{attribute 'no_check'}
// ModBus comunication master to multible slaves useing RTU protocol
// based on TF6255 - required lib: Tc2_ModbusRTU
FUNCTION_BLOCK ModbusRtuMaster22B
VAR_OUTPUT CONSTANT
	MIN_SLAVE												:	INT := 1;
	MAX_SLAVE												:	INT := PARAM.MODBUS_MAX_SLAVES_OF_MASTER;
{attribute 'displaymode':='binary'}
	OPTION_DISABLE_ERROR_STATE								:	BYTE := 2#0000_0001; //FB will not go into error state and keeps running, even all slaves are in error state
END_VAR
VAR_INPUT
	Enable													:	BOOL ; 		// FB will be processed as long as enable is TRUE 
	ResetTrig												:	BOOL ;		// The function block will be reset with a rising edge 
{attribute 'displaymode':='binary'}
	Options													:	BYTE := 0; //FB options, see VAR_OUTPUT CONSTANT
	SlaveCom												:	ARRAY[MIN_SLAVE..MAX_SLAVE] OF POINTER TO ModbusSlaveCom;
	Timestamp												:	DT;
END_VAR         	
VAR_OUTPUT     
	JobNo													:	INT := 0;
	SlaveNo													:	INT := 0;
{attribute 'displaymode':='binary'}
	SlaveInErrorMask										:	DWORD; //Bit.1 indicates slave 1 in error 	
	Error													:	BOOL;		// Rising edge of Error informs that an error occurred during the execution of the Function Block 
{attribute 'displaymode':='hex'}
	ErrorID													:	MODBUS_ERRORS;		// Error identification - see ADS return codes at Beckhoff infosys for further information 
	ErrorText												:	STRING;
END_VAR
VAR
(* memory **************************************************)
	State 													:	INT := 0;
(* trigger *************************************************)

(* timer ***************************************************)

(* blocks **************************************************)
//	com														:	ModbusRtuMaster_PcCOM := (Timeout := DEFAULT_ADS_TIMEOUT);
	com														:	ModbusRtuMaster_KL6x22B := (Timeout := DEFAULT_ADS_TIMEOUT);
//	com														:	ModbusRtuMaster_KL6x5B := (Timeout := DEFAULT_ADS_TIMEOUT);
(* internal used variables *********************************)
	i,j,k													:	INT :=0;
END_VAR

(* ModBus RTU comunication to multible slaves 	JHue V1.0			*)
(* uncomment necessary master funktion block 						*)
(* use TC2_ModBusRTU.lib											*)
(********************************************************************)

	IF ResetTrig THEN
		reset();
	END_IF
	
	CASE state OF
	0:	(* Idle *)
		IF Enable 
		THEN
			k 												:=	0;
			JobNo  :=  SlaveNo								:=	1;
			state 											:=	10;
		END_IF

	10: 
		IF GetNextSlave() 
		THEN (* find Slave *)
			k 												:= 0;
			IF GetNextJob() 
			THEN (* find JobNo *)
				SlaveCom[SlaveNo]^.currentJobIdx 			:= JobNo;
				SlaveCom[SlaveNo]^.writeJobRequested 		:= SlaveCom[SlaveNo]^.Jobs[JobNo].FunctionCode >= 5;
				State 										:= SEL(SlaveCom[SlaveNo]^.writeJobRequested, 20, 15);
			END_IF
		ELSE
			state 											:=	0;
		END_IF
	
	15: (* wait for valid write date *)
		IF NOT SlaveCom[SlaveNo]^.writeJobRequested
		THEN
			SlaveCom[SlaveNo]^.Jobs[JobNo].Valid 			:= FALSE;
			state 											:= 20;
		END_IF

	20: (* start job *)	
		IF NOT StartJob(FALSE) // Busy
		THEN						
			state 											:= 30;
		END_IF

	30: (* wait for com cycle *)
		IF NOT StartJob(TRUE) THEN // Not Busy, Execute set to True
			IF Error
			THEN
				ErrorText									:= CONCAT('Error at SlaveNo: ',	CONCAT(INT_TO_STRING(SlaveNo), CONCAT(', JobNo: ', INT_TO_STRING(JobNo))));
				SlaveCom[SlaveNo]^.countBad 				:= SlaveCom[SlaveNo]^.countBad +1;
				SlaveInErrorMask							:= CSETBIT32(SlaveInErrorMask,TO_SINT(SlaveNo),TRUE);
				IF Options.0
				THEN
					JobNo 									:= JobNo + 1;
					state 									:= 10;	(* next job *)				
				ELSE
					state 									:= 98; 					
				END_IF
			ELSE
				SlaveInErrorMask							:= CSETBIT32(SlaveInErrorMask,TO_SINT(SlaveNo),FALSE);
				SlaveCom[SlaveNo]^.countGood 				:= SlaveCom[SlaveNo]^.countGood +1;
				SlaveCom[SlaveNo]^.Jobs[JobNo].Valid 		:= TRUE;
				SlaveCom[SlaveNo]^.Jobs[JobNo].TimeStamp 	:= Timestamp;
				JobNo 										:= JobNo + 1;
				state 										:= 10;	(* next job *)
			END_IF
			StartJob(FALSE);
		END_IF

	98: (* wait for quit *)
		;


	END_CASE

METHOD PRIVATE getNextJob : Bool //Return value = TRUE if execution finished
VAR_INPUT
END_VAR
	
	WHILE SlaveCom[SlaveNo]^.Jobs[JobNo].FunctionCode = 0 DO
		JobNo 											:= JobNo + 1;
		IF JobNo > SlaveCom[SlaveNo]^.MAX_SLAVE_JOB THEN
			JobNo 										:= SlaveCom[SlaveNo]^.MIN_SLAVE_JOB;
			SlaveNo 									:= SlaveNo + 1;
			GetNextJob									:= FALSE;
			RETURN;
		END_IF
	END_WHILE
	GetNextJob											:= TRUE;
END_METHOD

METHOD PRIVATE getNextSlave : Bool //Return value = TRUE if execution finished
VAR_INPUT
END_VAR
	WHILE SlaveCom[SlaveNo] = 0 OR_ELSE NOT SlaveCom[SlaveNo]^.Enable DO
		SlaveNo 										:= SlaveNo + 1;
		IF SlaveNo > MAX_SLAVE 
		THEN
			k 											:= k + 1;
			SlaveNo 									:= MIN_SLAVE;
		ELSIF k = 2 
		THEN
			k 											:= 0;
			GetNextSlave								:= FALSE;
			RETURN;
		END_IF	
	END_WHILE
	GetNextSlave										:= TRUE;
END_METHOD

METHOD PUBLIC reset : BOOL //Return value = TRUE if execution finished
VAR_INPUT
END_VAR
IF State = 98 
THEN
	state													:= 0;
END_IF
Error														:= FALSE;
ErrorID														:= 0;
ErrorText													:= '';
reset														:= TRUE;
END_METHOD

METHOD PRIVATE startJob : BOOL //Return value = TRUE if busy - TRUE as long as the job is busy
VAR_INPUT
	Execute							: BOOL;
END_VAR
(* ModbusCOM Baustein mit parametern antriggern *)
	IF 	SlaveCom[SlaveNo]^.Jobs[JobNo].FunctionCode = 1 THEN
		com.ReadCoils(
			UnitID			:= SlaveCom[SlaveNo]^.Address,					(*UnitID: Modbus Stationsadresse (1..247). Der Modbus-Slave antwortet nur, wenn er Telegramme mit seiner eigenen Stationsadresse empfängt. optional können hier auch Sammeladressen eingestellt werden um auf beliebige Anfragen zu antworten. Die Adresse 0 ist für Broadcast-Telegramme reserviert und somit keine gültige Stationsadresse.*)
			Quantity		:= SlaveCom[SlaveNo]^.jobs[JobNo].Quantity,		(*Quantity: Anzahl der zu lesenden oder zu schreibenden Datenworte bei Wort-orientierten Modbus-Funktionen. Bei Bit-orientierten Modbus-Funktionen gibt Quantity die Anzahl der Bits (Inputs oder Coils) an.*)
			MBAddr			:= SlaveCom[SlaveNo]^.jobs[JobNo].startAddress,	(*MBAddr: Modbus-Datenadresse, von der die Daten aus dem Endgerät (Slave) gelesen werden. Diese Adresse wird unverändert zum Slave übertragen und wird dort als Datenadresse interpretiert.*)
			cbLength		:= SlaveCom[SlaveNo]^.jobs[JobNo].Quantity, 	(*cbLength : Größe der verwendeten Datenvariable für Sende- oder Lese-Aktionen in Bytes. cbLength muss größer oder gleich der durch Quantity bestimmten übertragenen Datenmenge sein. Bei Wortzugriffen gilt z. B.: [cbLength >= Quantity * 2]. cbLength kann mit SIZEOF(ModbusDaten) berechnet werden.*)
			pMemoryAddr		:= ADR(SlaveCom[SlaveNo]^.Data),				(*pMemoryAddr: Speicheradresse in der SPS, die mit ADR(ModbusDaten) berechnet wird. Bei Leseaktionen werden die gelesenen Daten in der adressierten Variablen abgelegt. Bei Sende-Aktionen werden die Daten aus der adressierten Variablen zum Endgerät übertragen.*)
			Execute			:= Execute,
			Timeout			:= ,
			BUSY			=> StartJob,									(*Busy: Zeigt an, dass der Funktionsbaustein aktiv ist. Busy wird mit steigender Flanke an Execute TRUE und wird wieder FALSE nachdem die gestartete Aktion beendet ist. Es kann immer nur eine Aktion gleichzeitig aktiv sein.*)
			Error			=> Error,										(*Error: Zeigt an, dass bei der Bearbeitung einer Aktion ein Fehler aufgetreten ist*)
			ErrorId			=> ErrorID);									(*ErrorId: Zeigt eine Fehlernummer im Falle einer gestörten oder fehlerhaften Kommunikation an.*)	

	ELSIF 	SlaveCom[SlaveNo]^.Jobs[JobNo].FunctionCode = 3 THEN
		com.ReadRegs(
			UnitID			:= SlaveCom[SlaveNo]^.Address,		
			Quantity		:= SlaveCom[SlaveNo]^.jobs[JobNo].Quantity,
			MBAddr			:= SlaveCom[SlaveNo]^.jobs[JobNo].startAddress,
			cbLength		:= SlaveCom[SlaveNo]^.jobs[JobNo].Quantity * 2,
			pMemoryAddr		:= ADR(SlaveCom[SlaveNo]^.data),
			Execute			:= Execute,
			Timeout			:= ,
			BUSY			=> StartJob,
			Error			=> Error,
			ErrorId			=> ErrorID);
	
	ELSIF 	SlaveCom[SlaveNo]^.Jobs[JobNo].FunctionCode = 4 THEN
		com.ReadInputRegs(
			UnitID			:= SlaveCom[SlaveNo]^.Address,		
			Quantity		:= SlaveCom[SlaveNo]^.jobs[JobNo].Quantity,
			MBAddr			:= SlaveCom[SlaveNo]^.jobs[JobNo].startAddress,
			cbLength		:= SlaveCom[SlaveNo]^.jobs[JobNo].Quantity * 2,
			pMemoryAddr		:= ADR(SlaveCom[SlaveNo]^.data),
			Execute			:= Execute,
			Timeout			:= ,
			BUSY			=> StartJob,
			Error			=> Error,
			ErrorId			=> ErrorID);
	
	ELSIF 	SlaveCom[SlaveNo]^.Jobs[JobNo].FunctionCode = 5 THEN
		com.WriteSingleCoil(
			UnitID			:= SlaveCom[SlaveNo]^.Address,		
			Quantity		:= SlaveCom[SlaveNo]^.jobs[JobNo].Quantity,
			MBAddr			:= SlaveCom[SlaveNo]^.jobs[JobNo].startAddress,
			cbLength		:= SlaveCom[SlaveNo]^.jobs[JobNo].Quantity,
			pMemoryAddr		:= ADR(SlaveCom[SlaveNo]^.data),
			Execute			:= Execute,
			Timeout			:= ,
			BUSY			=> StartJob,
			Error			=> Error,
			ErrorId			=> ErrorID);
			
	ELSIF 	SlaveCom[SlaveNo]^.Jobs[JobNo].FunctionCode = 6 THEN
		com.WriteSingleRegister(
			UnitID			:= SlaveCom[SlaveNo]^.Address,		
			Quantity		:= SlaveCom[SlaveNo]^.jobs[JobNo].Quantity,
			MBAddr			:= SlaveCom[SlaveNo]^.jobs[JobNo].startAddress,
			cbLength		:= SlaveCom[SlaveNo]^.jobs[JobNo].Quantity,
			pMemoryAddr		:= ADR(SlaveCom[SlaveNo]^.data),
			Execute			:= Execute,
			Timeout			:= ,
			BUSY			=> StartJob,
			Error			=> Error,
			ErrorId			=> ErrorID);
		
	ELSIF 	SlaveCom[SlaveNo]^.Jobs[JobNo].FunctionCode = 8 THEN
		com.Diagnostics(
			UnitID			:= SlaveCom[SlaveNo]^.Address,		
			Quantity		:= SlaveCom[SlaveNo]^.jobs[JobNo].Quantity,
			MBAddr			:= SlaveCom[SlaveNo]^.jobs[JobNo].startAddress,
			cbLength		:= SlaveCom[SlaveNo]^.jobs[JobNo].Quantity,
			pMemoryAddr		:= ADR(SlaveCom[SlaveNo]^.data),
			Execute			:= Execute,
			Timeout			:= ,
			BUSY			=> StartJob,
			Error			=> Error,
			ErrorId			=> ErrorID);
		
	ELSIF 	SlaveCom[SlaveNo]^.Jobs[JobNo].FunctionCode = 15 THEN
		com.WriteMultipleCoils(
			UnitID			:= SlaveCom[SlaveNo]^.Address,		
			Quantity		:= SlaveCom[SlaveNo]^.jobs[JobNo].Quantity,
			MBAddr			:= SlaveCom[SlaveNo]^.jobs[JobNo].startAddress,
			cbLength		:= SlaveCom[SlaveNo]^.jobs[JobNo].Quantity,
			pMemoryAddr		:= ADR(SlaveCom[SlaveNo]^.data),
			Execute			:= Execute,
			Timeout			:= ,
			BUSY			=> StartJob,
			Error			=> Error,
			ErrorId			=> ErrorID);
	
	ELSIF 	SlaveCom[SlaveNo]^.Jobs[JobNo].FunctionCode = 16 THEN
		com.WriteRegs(
			UnitID			:= SlaveCom[SlaveNo]^.Address,		
			Quantity		:= SlaveCom[SlaveNo]^.jobs[JobNo].Quantity,
			MBAddr			:= SlaveCom[SlaveNo]^.jobs[JobNo].startAddress,
			cbLength		:= SlaveCom[SlaveNo]^.jobs[JobNo].Quantity,
			pMemoryAddr		:= ADR(SlaveCom[SlaveNo]^.data),
			Execute			:= Execute,
			Timeout			:= ,
			BUSY			=> StartJob,
			Error			=> Error,
			ErrorId			=> ErrorID);
			
	END_IF
END_METHOD

END_FUNCTION_BLOCK

(* stored: Version 1.1.0.1, ProductVersion 3.1.4024.16
   POU ModbusRtuMaster22B: Id {845e89ad-8649-4d53-8a66-85f39e98e6ac}, SpecialFunc None
   Method getNextJob: Id {0ece9eb7-bffb-4bf4-92ff-dda6a1efe828}
   Method getNextSlave: Id {89f1f579-488d-468b-a088-d0c1af208ce5}
   Method reset: Id {257589db-cb94-42d5-be03-34c2530682ed}
   Method startJob: Id {745ddb85-e7e4-4570-b217-29a3bcee8fff} *)
